TYPE UA_OptionSet :
STRUCT
END_STRUCT
END_TYPE

(* stored: Version 1.1.0.1
   DUT UA_OptionSet: Id {82e5dae4-ebae-433d-9345-e1f8104b90c3} *)
